{attribute 'GeneratedUsingTerminal: EL3443-0000-0016'}
{attribute addProperty BoxType "EL3443-0000-0016"}
{attribute addProperty Id "FrequencyAT %I*REAL4Power_FactorAT %I*REAL4Calculated_Neutral_Line_CurrentAT %I*REAL4"}
{attribute addProperty CRC "4230807319"}
{attribute addProperty Size "12"}
TYPE Total_Basic_FC2CFF17 :
STRUCT
	{attribute addProperty Name "Frequency"}
	Frequency AT %I* : REAL;
	{attribute addProperty Name "Power_Factor"}
	Power_Factor AT %I* : REAL;
	{attribute addProperty Name "Calculated_Neutral_Line_Current"}
	Calculated_Neutral_Line_Current AT %I* : REAL;
END_STRUCT
END_TYPE

(* stored: Version 1.2.0.0, ProductVersion 3.1.4024.9
   DUT Total_Basic_FC2CFF17: Id {4b20edd9-5970-4e12-af47-6d2fc8625f90} *)
